GLOBALCONSTANTS DefaultPool (* Global constants *)
  PACKAGE Uebungen::const::UT;
  VAR_GLOBAL CONSTANT
    ISO_DESIGNATOR_WIDTH : UINT := 80;
    ISO_DESIGNATOR_HEIGHT : UINT := 80;
    ISO_MASK_SIZE : UINT := 480;
    ISO_VERSION_LABEL : STRING;
    MASK_WIDTH : UINT := 480;
    MASK_HEIGHT : UINT := 480;
    WorkingSet : UINT := 0;
    Macro_Go_To_DataMask_M1 : UINT := 1;
    Macro_Go_To_DataMask_M2 : UINT := 2;
    Macro_Go_To_DataMask_M3 : UINT := 3;
    DataMask_M1 : UINT := 1000;
    DataMask_M2 : UINT := 1001;
    DataMask_M3 : UINT := 1002;
    AlarmMask_A1_low : UINT := 2000;
    AlarmMask_A2_medium : UINT := 2001;
    AlarmMask_A3_high : UINT := 2002;
    Container_B : UINT := 3000;
    Container_low : UINT := 3001;
    Container_medium : UINT := 3002;
    Container_high : UINT := 3003;
    SoftKeyMask_S1 : UINT := 4000;
    SoftKey_F1 : UINT := 5000;
    SoftKey_F2 : UINT := 5001;
    SoftKey_F3 : UINT := 5002;
    SoftKey_F4 : UINT := 5003;
    SoftKey_F5 : UINT := 5004;
    SoftKey_F6 : UINT := 5005;
    SoftKey_F7 : UINT := 5006;
    SoftKey_F8 : UINT := 5007;
    SoftKey_F9 : UINT := 5008;
    SoftKey_F10 : UINT := 5009;
    SoftKey_F11 : UINT := 5010;
    SoftKey_F12 : UINT := 5011;
    Button_A1 : UINT := 6000;
    Button_A2 : UINT := 6001;
    Button_L1 : UINT := 6002;
    Button_A3 : UINT := 6003;
    InputString_S1 : UINT := 8000;
    InputNumber_I1 : UINT := 9000;
    InputNumber_I2 : UINT := 9001;
    InputNumber_I3 : UINT := 9002;
    InputNumber_I4 : UINT := 9003;
    OutputString_WorkingSet_0 : UINT := 11000;
    OutputString_SoftKey_F1 : UINT := 11001;
    OutputString_SoftKey_F2 : UINT := 11002;
    OutputString_SoftKey_F3 : UINT := 11003;
    OutputString_SoftKey_F4 : UINT := 11004;
    OutputString_SoftKey_F5 : UINT := 11005;
    OutputString_SoftKey_F6 : UINT := 11006;
    OutputString_SoftKey_F7 : UINT := 11007;
    OutputString_SoftKey_F8 : UINT := 11008;
    OutputString_SoftKey_F9 : UINT := 11009;
    OutputString_SoftKey_F10 : UINT := 11010;
    OutputString_SoftKey_F11 : UINT := 11011;
    OutputString_SoftKey_F12 : UINT := 11012;
    OutputString_DataMask_M1 : UINT := 11013;
    OutputString_DataMask_M2 : UINT := 11014;
    OutputString_Go_To_DataMask_M1 : UINT := 11015;
    OutputString_Go_To_DataMask_M2 : UINT := 11016;
    OutputString_Button_A1 : UINT := 11017;
    OutputString_Button_A2 : UINT := 11018;
    OutputString_OutputNumber_N1 : UINT := 11019;
    OutputString_OutputNumber_N2 : UINT := 11020;
    OutputString_InputNumber_I1 : UINT := 11021;
    OutputString_InputNumber_I2 : UINT := 11022;
    OutputString : UINT := 11023;
    OutputString_Button_L1 : UINT := 11024;
    OutputString_InputString_S1 : UINT := 11025;
    OutputString_Go_To_DataMask_M3 : UINT := 11026;
    OutputString_Button_A3 : UINT := 11027;
    OutputString_InputNumber_I3 : UINT := 11028;
    OutputString_InputNumber_I4 : UINT := 11029;
    OutputString_OutputNumber_N3 : UINT := 11030;
    OutputNumber_N1 : UINT := 12000;
    OutputNumber_N2 : UINT := 12001;
    OutputNumber_N3 : UINT := 12002;
    Line_W : UINT := 13000;
    Line_S : UINT := 13001;
    Rectangle_black : UINT := 14000;
    Rectangle_grey : UINT := 14001;
    Rectangle_yellow : UINT := 14002;
    Rectangle_red : UINT := 14003;
    information : UINT := 20001;
    alert : UINT := 20002;
    Caution : UINT := 20003;
    Meisterschulen_LogoG1_256 : UINT := 20004;
    Logos_icon : UINT := 20500;
    FontAttributes_6x8 : UINT := 23000;
    FontAttributes_8x12 : UINT := 23001;
    FontAttributes_12x16 : UINT := 23002;
    LineAttributes_black : UINT := 24000;
    LineAttributes_black_3 : UINT := 24001;
    LineAttributes_grey_3 : UINT := 24002;
    LineAttributes_yellow_3 : UINT := 24003;
    LineAttributes_red_3 : UINT := 24004;
    FillAttributes_white : UINT := 25000;
    ObjectPointer_P1 : UINT := 27000;
    AuxFunction2_X1 : UINT := 31000;
  END_VAR
END_GLOBALCONSTANTS
